FUNCTION_BLOCK GET_AT_INDEX (* Service Interface Function Block Type *)
  (* Standard: 61499-2; Description: Fetch value from array at given index. Array data type has to match with output data type. *)
  (* Version 0.0, 2014-07-11, Matthias Plasch, 4DIAC-Consortium *)
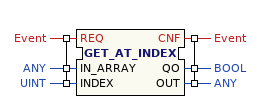
  EVENT_INPUT
    REQ WITH IN_ARRAY, INDEX; (* Service Request *)
  END_EVENT
  EVENT_OUTPUT
    CNF WITH QO, OUT; (* Confirmation of Requested Service *)
  END_EVENT
  VAR_INPUT
    IN_ARRAY : ANY; (* input array *)
    INDEX : UINT; (* index to fetch value from *)
  END_VAR
  VAR_OUTPUT
    QO : BOOL; (* Event Output Qualifier *)
    OUT : ANY; (* fetched output value *)
  END_VAR
  (* Service APPLICATION/RESOURCE: Service Interface Function Block Type *)
END_FUNCTION_BLOCK
